TYPE ST_DCSystemDefaultParameters :
STRUCT
	aSetPointLimitsTemperature : ARRAY[1..2] OF REAL := [20,40];
END_STRUCT
END_TYPE

(* stored: Version 1.1.0.1, ProductVersion 3.1.4024.10
   DUT ST_DCSystemDefaultParameters: Id {496e80cc-a8e2-48d6-803b-19682b772885} *)
